function_block FINAL FB_Syntax_Final extends FB_Syntax_Derived var _nValue    : int; end_var

_nValue := _nValue + 1;

END_FUNCTION_BLOCK

(* stored: Version 1.1.0.1, ProductVersion 3.1.4024.16
   POU FB_Syntax_Final: Id {2d0a4735-e35b-4a3e-a618-594a67464bce}, SpecialFunc None *)
